// Tries to guess if the given pointer refers to a function block instance. 
// [note] 
// This is heuristic and can be inaccurate. For reliable checks, the FB 
// must implement __SYSTEM.IQueryInterface. If the FB does not implement
// IQueryInterface, its type cannot be safely determined.
FUNCTION F_IsFunctionBlock : BOOL // TRUE if pointer appears to be a function block instance.
VAR_INPUT
	// Pointer to test.
	pValue : POINTER TO BYTE;
END_VAR
VAR
	pCheck : POINTER TO __UXINT;
END_VAR

pCheck := pValue;

CASE F_GetAddressMemoryArea(pCheck) OF 
	E_AddressMemoryArea.Static,
	E_AddressMemoryArea.Dynamic:
		pCheck := pCheck^;
ELSE
	RETURN;
	END_CASE
	
CASE F_GetAddressMemoryArea(pCheck) OF 
	E_AddressMemoryArea.Static,
	E_AddressMemoryArea.Dynamic:
		F_IsFunctionBlock := pCheck^ = SIZEOF(__UXINT);
	END_CASE

END_FUNCTION

(* stored: Version 1.1.0.1
   POU F_IsFunctionBlock: Id {90f7e604-cf59-0534-075a-85679a02d1bc}, SpecialFunc None *)
